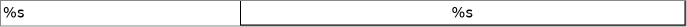
VISUALIZATION VISU_ProcessStep  // 687x27
VAR_IN_OUT
	widget : ProcessStepWidget;
END_VAR
    Rectangle (240,0 445x25), "%s", text variable: widget.statusText, invisible if: widget.inivisible, colour variable: widget.color.bg
        p3450524324: widget.color.fg
        p55702900: widget.color.fg
    Rectangle (0,0 235x25), "%s", text variable: widget.description, invisible if: widget.inivisible
END_VISUALIZATION

(* stored: Version 1.1.0.1, ProductVersion 3.1.4018.5
   Visu VISU_ProcessStep: Id {b61c9714-0ed1-49b5-8beb-aedd07886fe0} *)
